// Mitsubishi GX Works2 project: 생자연습001   PLC: Q03UDE

// global labels: Global1
VAR_GLOBAL
  PB1 AT X0 : BOOL;
  PB2 AT X1 : BOOL;
  PB3 AT X2 : BOOL;
  TG_SW AT X3 : BOOL;
  S1센서 AT X8 : BOOL;
  S3고주파 AT X9 : BOOL;
  S4용량형 AT X0A : BOOL;
  공급전 AT X10 : BOOL;
  공급후 AT X11 : BOOL;
  가공전 AT X12 : BOOL;
  가공후 AT X13 : BOOL;
  송출전 AT X14 : BOOL;
  송출후 AT X15 : BOOL;
  배출전 AT X16 : BOOL;
  배출후 AT X17 : BOOL;
  공급전솔 AT Y20 : BOOL;
  공급후솔 AT Y21 : BOOL;
  송출전솔 AT Y22 : BOOL;
  송출후솔 AT Y23 : BOOL;
  배출전솔 AT Y24 : BOOL;
  배출후솔 AT Y25 : BOOL;
  가공전솔 AT Y26 : BOOL;
  가공드릴 AT Y27 : BOOL;
  CON_CW AT Y28 : BOOL;
  적색램프 AT Y30 : BOOL;
  황색램프 AT Y31 : BOOL;
  녹색램프 AT Y32 : BOOL;
END_VAR

PROGRAM MAIN
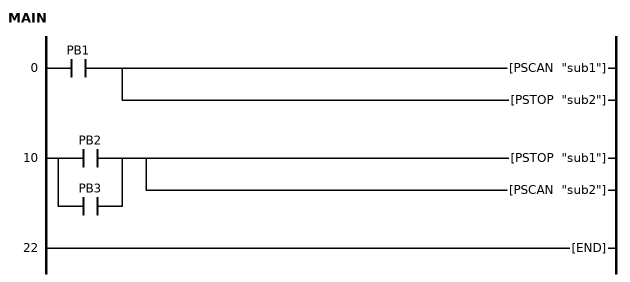
0     LD      PB1
      PSCAN   "sub1"
      PSTOP   "sub2"
10    LD      PB2
      OR      PB3
      PSTOP   "sub1"
      PSCAN   "sub2"
22    END
END_PROGRAM

PROGRAM sub1
VAR
  공급전진 : BOOL;
  송출전진 : BOOL;
  배출전진 : BOOL;
  T지연 : TIMER;
  송출후진 : BOOL;
  가공전진 : BOOL;
  가공후진 : BOOL;
  공급후진 : BOOL;
  배출후진 : BOOL;
  기본종료 : BOOL;
END_VAR
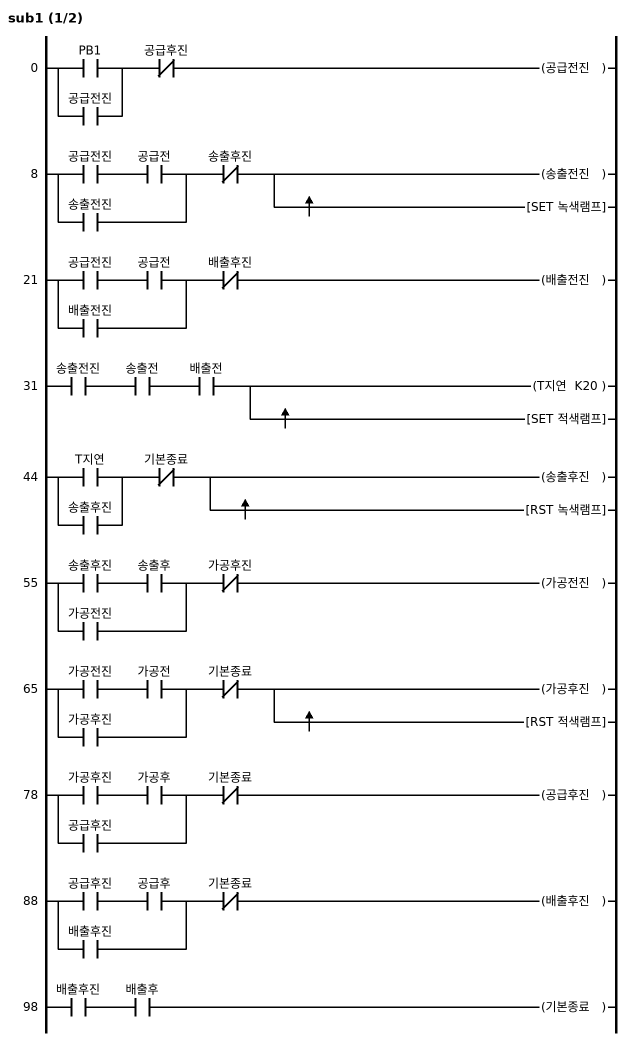
0     LD      PB1
      OR      공급전진
      ANI     공급후진
      OUT     공급전진
8     LD      공급전진
      AND     공급전
      OR      송출전진
      ANI     송출후진
      OUT     송출전진
      MEP
      SET     녹색램프
21    LD      공급전진
      AND     공급전
      OR      배출전진
      ANI     배출후진
      OUT     배출전진
31    LD      송출전진
      AND     송출전
      AND     배출전
      OUT     T지연 K20
      MEP
      SET     적색램프
44    LD      T지연
      OR      송출후진
      ANI     기본종료
      OUT     송출후진
      MEP
      RST     녹색램프
55    LD      송출후진
      AND     송출후
      OR      가공전진
      ANI     가공후진
      OUT     가공전진
65    LD      가공전진
      AND     가공전
      OR      가공후진
      ANI     기본종료
      OUT     가공후진
      MEP
      RST     적색램프
78    LD      가공후진
      AND     가공후
      OR      공급후진
      ANI     기본종료
      OUT     공급후진
88    LD      공급후진
      AND     공급후
      OR      배출후진
      ANI     기본종료
      OUT     배출후진
98    LD      배출후진
      AND     배출후
      OUT     기본종료
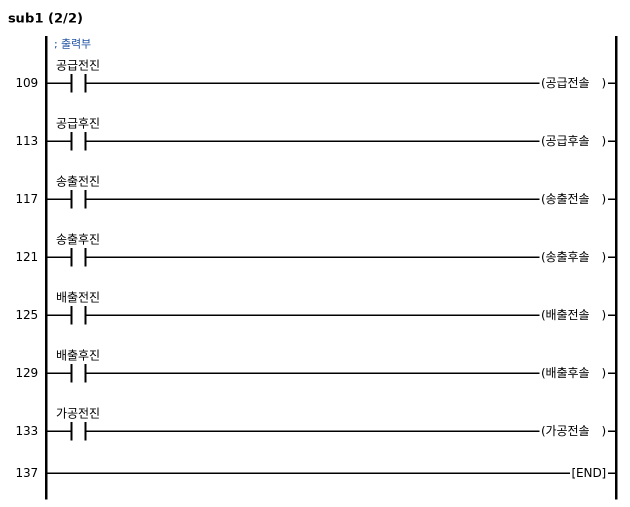
; 출력부
109   LD      공급전진
      OUT     공급전솔
113   LD      공급후진
      OUT     공급후솔
117   LD      송출전진
      OUT     송출전솔
121   LD      송출후진
      OUT     송출후솔
125   LD      배출전진
      OUT     배출전솔
129   LD      배출후진
      OUT     배출후솔
133   LD      가공전진
      OUT     가공전솔
137   END
END_PROGRAM

PROGRAM sub2
VAR
  공급전진 : BOOL;
  드릴온 : BOOL;
  가공전진 : BOOL;
  가공후진 : BOOL;
  드릴오프 : BOOL;
  공급후진 : BOOL;
  송출전진 : BOOL;
  송출후진 : BOOL;
  컨구동 : BOOL;
  금속탐지 : BOOL;
  비금속탐지 : BOOL;
  T금속지연 : TIMER;
  배출전진 : BOOL;
  배출후진 : BOOL;
  금종 : BOOL;
  T비금속지연 : TIMER;
  비종 : BOOL;
  종료 : BOOL;
  연속시작 : BOOL;
  연속공정 : BOOL;
  C금속 : COUNTER;
  T초기화리셋 : TIMER;
END_VAR
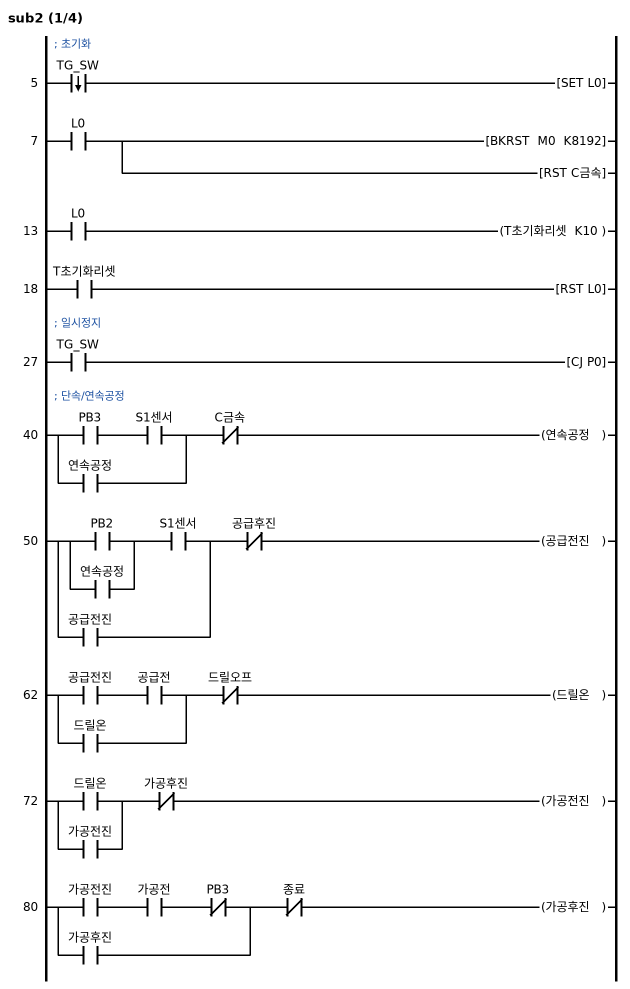
; 초기화
5     LDF     TG_SW
      SET     L0
7     LD      L0
      BKRST   M0 K8192
      RST     C금속
13    LD      L0
      OUT     T초기화리셋 K10
18    LD      T초기화리셋
      RST     L0
; 일시정지
27    LD      TG_SW
      CJ      P0
; 단속/연속공정
40    LD      PB3
      AND     S1센서
      OR      연속공정
      ANI     C금속
      OUT     연속공정
50    LD      PB2
      OR      연속공정
      AND     S1센서
      OR      공급전진
      ANI     공급후진
      OUT     공급전진
62    LD      공급전진
      AND     공급전
      OR      드릴온
      ANI     드릴오프
      OUT     드릴온
72    LD      드릴온
      OR      가공전진
      ANI     가공후진
      OUT     가공전진
80    LD      가공전진
      AND     가공전
      ANI     PB3
      OR      가공후진
      ANI     종료
      OUT     가공후진
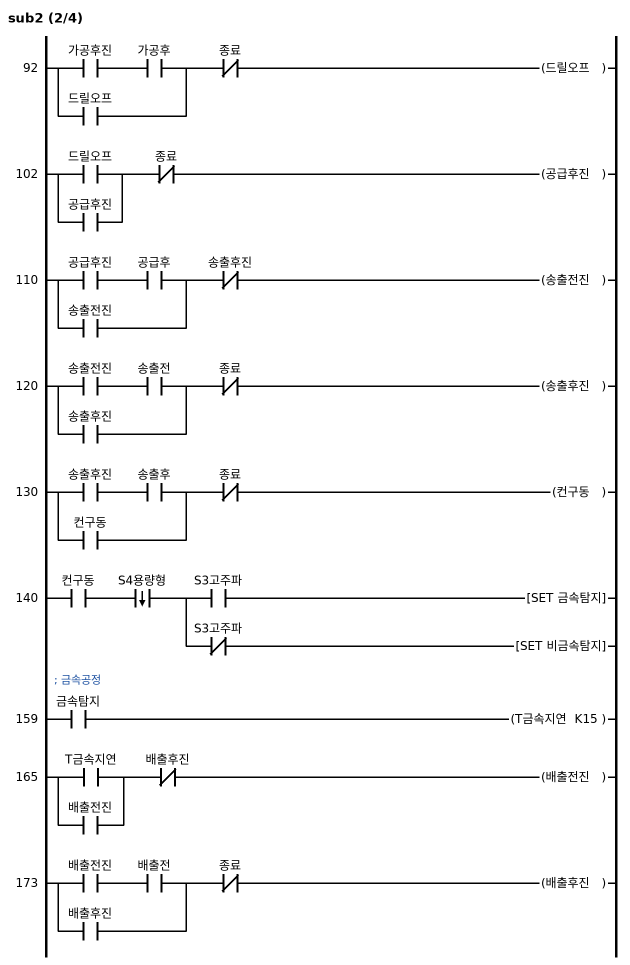
92    LD      가공후진
      AND     가공후
      OR      드릴오프
      ANI     종료
      OUT     드릴오프
102   LD      드릴오프
      OR      공급후진
      ANI     종료
      OUT     공급후진
110   LD      공급후진
      AND     공급후
      OR      송출전진
      ANI     송출후진
      OUT     송출전진
120   LD      송출전진
      AND     송출전
      OR      송출후진
      ANI     종료
      OUT     송출후진
130   LD      송출후진
      AND     송출후
      OR      컨구동
      ANI     종료
      OUT     컨구동
140   LD      컨구동
      ANDF    S4용량형
      MPS
      AND     S3고주파
      SET     금속탐지
      MPP
      ANI     S3고주파
      SET     비금속탐지
; 금속공정
159   LD      금속탐지
      OUT     T금속지연 K15
165   LD      T금속지연
      OR      배출전진
      ANI     배출후진
      OUT     배출전진
173   LD      배출전진
      AND     배출전
      OR      배출후진
      ANI     종료
      OUT     배출후진
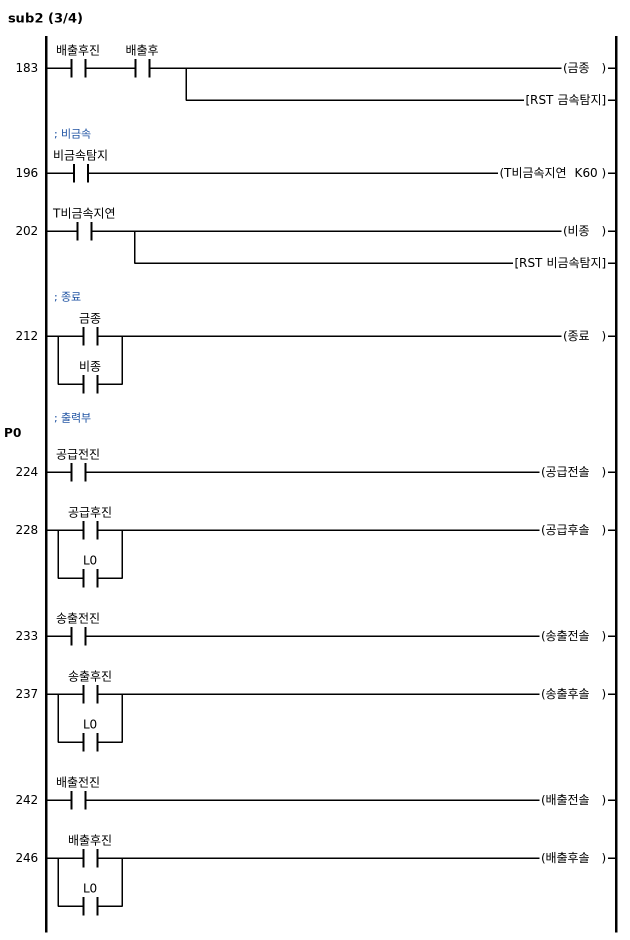
183   LD      배출후진
      AND     배출후
      OUT     금종
      RST     금속탐지
; 비금속
196   LD      비금속탐지
      OUT     T비금속지연 K60
202   LD      T비금속지연
      OUT     비종
      RST     비금속탐지
; 종료
212   LD      금종
      OR      비종
      OUT     종료
; 출력부
      P0
224   LD      공급전진
      OUT     공급전솔
228   LD      공급후진
      OR      L0
      OUT     공급후솔
233   LD      송출전진
      OUT     송출전솔
237   LD      송출후진
      OR      L0
      OUT     송출후솔
242   LD      배출전진
      OUT     배출전솔
246   LD      배출후진
      OR      L0
      OUT     배출후솔
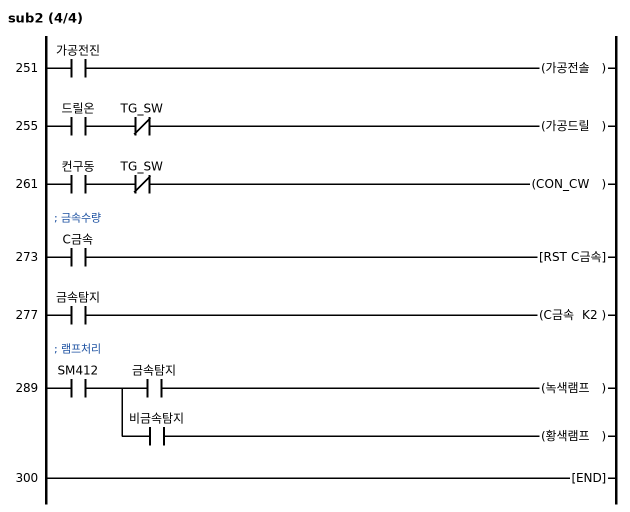
251   LD      가공전진
      OUT     가공전솔
255   LD      드릴온
      ANI     TG_SW
      OUT     가공드릴
261   LD      컨구동
      ANI     TG_SW
      OUT     CON_CW
; 금속수량
273   LD      C금속
      RST     C금속
277   LD      금속탐지
      OUT     C금속 K2
; 램프처리
289   LD      SM412
      MPS
      AND     금속탐지
      OUT     녹색램프
      MPP
      AND     비금속탐지
      OUT     황색램프
300   END
END_PROGRAM
